FUNCTION_BLOCK CALIBRATE_3P (* BOOL-triggered 3-point calibration for joysticks (Min, Mid, Max) *)
  (* Standard: 61499-1 *)
  (* Version 1.0, 2026-06-01, Meisterschulen am Ostbahnhof *)
  PACKAGE OSCAT::Basic::POUs::Engineering::measurements;
  (* Documentation:
  Formula
    Y = piecewise linear interpolation between stored calibration points Calibration (3-Point)
    - Min (C_MIN=TRUE): Move joystick to minimum position, set C_MIN=TRUE
   X_MIN := X → stores current raw value as Min point
   - Mid (C_MID=TRUE): Move joystick to center, set C_MID=TRUE
   X_MID := X → stores current raw value as Mid point (center)
   - Max (C_MAX=TRUE): Move joystick to maximum position, set C_MAX=TRUE
   X_MAX := X → stores current raw value as Max point
    Note: The calibration points can be calibrated in any order and can be repeated individually. Only one point per REQ event (ELSIF chain).
   Output Calculation
    - If X < X_MID: linear interpolation between (X_MIN, MIN_REF) and (X_MID, MID_REF)
   - If X >= X_MID: linear interpolation between (X_MID, MID_REF) and (X_MAX, MAX_REF)
   - Output is clipped to MIN_REF..MAX_REF
    Example
   Scenario: Joystick with center drift. Raw range 0..1000, desired output -100..0..100.
      Step |  Action |  Result |  
    1 |  Move joystick to min, set C_MIN=TRUE |  X_MIN = 50 (drifted from ideal 0) |  
    2 |  Move joystick to center, set C_MID=TRUE |  X_MID = 520 (drifted from ideal 500) |  
    3 |  Move joystick to max, set C_MAX=TRUE |  X_MAX = 980 (drifted from ideal 1000) |  
     Output: Interpolated between MIN_REF=-100, MID_REF=0, MAX_REF=100 with clipping.
  *)
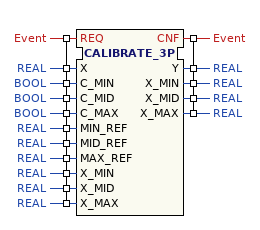
  EVENT_INPUT
    REQ WITH X, C_MIN, C_MID, C_MAX, MIN_REF, MID_REF, MAX_REF, X_MIN, X_MID, X_MAX; (* Normal Execution Request *)
  END_EVENT
  EVENT_OUTPUT
    CNF WITH Y, X_MIN, X_MID, X_MAX; (* Execution Confirmation *)
  END_EVENT
  VAR_INPUT
    X : REAL; (* Raw Input *)
    C_MIN : BOOL; (* Calibrate Min Point *)
    C_MID : BOOL; (* Calibrate Mid Point (Center) *)
    C_MAX : BOOL; (* Calibrate Max Point *)
    MIN_REF : REAL := 0.0; (* Target value for Min *)
    MID_REF : REAL := 50.0; (* Target value for Mid *)
    MAX_REF : REAL := 100.0; (* Target value for Max *)
  END_VAR
  VAR_OUTPUT
    Y : REAL; (* Calibrated Output *)
  END_VAR
  VAR_IN_OUT
    X_MIN : REAL := 0.0; (* Stored Min Value *)
    X_MID : REAL := 50.0; (* Stored Mid Value *)
    X_MAX : REAL := 100.0; (* Stored Max Value *)
  END_VAR
  EC_STATES
    REQ : REQ -> CNF;
  END_STATES
  ALGORITHM REQ IN ST:
(* calibration: store current raw input for the active point *)
IF C_MIN THEN
	X_MIN := X;
ELSIF C_MID THEN
	X_MID := X;
ELSIF C_MAX THEN
	X_MAX := X;
END_IF;

(* piecewise linear interpolation between stored calibration points *)
IF X < X_MID THEN
	IF X_MID > X_MIN THEN
		Y := MIN_REF + (X - X_MIN) * (MID_REF - MIN_REF) / (X_MID - X_MIN);
	ELSE
		Y := MIN_REF;
	END_IF;
ELSE
	IF X_MAX > X_MID THEN
		Y := MID_REF + (X - X_MID) * (MAX_REF - MID_REF) / (X_MAX - X_MID);
	ELSE
		Y := MID_REF;
	END_IF;
END_IF;

(* clip output to reference range *)
IF Y < MIN_REF THEN
	Y := MIN_REF;
ELSIF Y > MAX_REF THEN
	Y := MAX_REF;
END_IF;
  END_ALGORITHM
END_FUNCTION_BLOCK
